{attribute 'qualified_only'}
VAR_GLOBAL
	testString : STRING;
	
END_VAR

(* stored: Version 1.1.0.1, ProductVersion 3.1.4024.12
   GVL GVL: Id {a5c1b19b-d0f5-4110-b3d5-d335b4733d12} *)
